(* PLC project JSR_Sample_10062022.ecp, WAGO e!COCKPIT e!COCKPIT *)
(* stored: creationDateTime 2022-10-12T15:24:50.162515, modificationDateTime 2022-10-12T15:16:09.7000612 *)

FUNCTION_BLOCK fb_SMC_EX260
  VAR_INPUT
    sInput1 : SINT;  (* SMC Inputs *)
    bInput2 : BYTE;
    xOutA : ARRAY[1..16] OF BOOL;  (* Program Outputs *)
    xOutB : ARRAY[1..16] OF BOOL;
  END_VAR
  VAR_OUTPUT
    sOutput1 : SINT;  (* SMC Outputs *)
    bOutput2 : BYTE;
    bOutput3 : BYTE;
    bOutput4 : BYTE;
  END_VAR

            sOutput1.0 := xOutA[1];
sOutput1.1 := xOutB[1];
sOutput1.2 := xOutA[2];
sOutput1.3 := xOutB[2];
sOutput1.4 := xOutA[3];
sOutput1.5 := xOutB[3];
sOutput1.6 := xOutA[4];
sOutput1.7 := xOutB[4];

bOutput2.0 := xOutA[5];
bOutput2.1 := xOutB[5];
bOutput2.2 := xOutA[6];
bOutput2.3 := xOutB[6];
bOutput2.4 := xOutA[7];
bOutput2.5 := xOutB[7];
bOutput2.6 := xOutA[8];
bOutput2.7 := xOutB[8];

bOutput3.0 := xOutA[9];
bOutput3.1 := xOutB[9];
bOutput3.2 := xOutA[10];
bOutput3.3 := xOutB[10];
bOutput3.4 := xOutA[11];
bOutput3.5 := xOutB[11];
bOutput3.6 := xOutA[12];
bOutput3.7 := xOutB[12];

bOutput4.0 := xOutA[13];
bOutput4.1 := xOutB[13];
bOutput4.2 := xOutA[14];
bOutput4.3 := xOutB[14];
bOutput4.4 := xOutA[15];
bOutput4.5 := xOutB[15];
bOutput4.6 := xOutA[16];
bOutput4.7 := xOutB[16];

          
END_FUNCTION_BLOCK
